// TwinCAT 3 PLC project PLC_1
// ProgramVersion: 3.1.4023.0
// libraries:
//   Tc2_ModbusRTU, * (Beckhoff Automation GmbH)
//   Tc2_Standard, * (Beckhoff Automation GmbH)
//   Tc2_System, * (Beckhoff Automation GmbH)
//   Tc3_Module, * (Beckhoff Automation GmbH)
// project tree:
//   / PlcTask.TcTTO
//   POUs/ MAIN.TcPOU, POU_Mdbus.TcPOU
// real-time tasks:
//   TASK PlcTask: cycle T#10ms, priority 20, ADS port 350

CONFIGURATION PLC_1
    RESOURCE PLC ON TwinCAT3
        TASK PlcTask(INTERVAL := T#10ms, PRIORITY := 20);
        PROGRAM MAIN WITH PlcTask : MAIN;
    END_RESOURCE
END_CONFIGURATION

// ---- POUs/MAIN.TcPOU
PROGRAM MAIN
VAR
END_VAR

POU_Mdbus();

END_PROGRAM

// ---- POUs/POU_Mdbus.TcPOU
PROGRAM POU_Mdbus
VAR
    fbModbusRead : FB_MBReadRegs ;
    fbModbusWrite : FB_MBWriteRegs ;
     
    iStep: INT;
     
    aModbusRead : ARRAY[1..10] OF INT ;
    aModbusWrite : ARRAY[1..10] OF INT ;    
END_VAR

CASE iStep OF
    0:
        fbModbusRead(bExecute:= FALSE );
        fbModbusWrite(bExecute := FALSE);       
        iStep := 10 ;
     
     
    10 : 
        fbModbusRead(
            sIPAddr:= '192.168.2.102', 
            nTCPPort:= 502, 
            nUnitID:= 255, 
            nQuantity:= 10, 
            nMBAddr:= 8000, 
            cbLength:= SIZEOF(aModbusRead), 
            pDestAddr:= ADR(aModbusRead), 
            bExecute:= TRUE, 
            tTimeout:= T#2S, 
            bBusy=> , 
            bError=> , 
            nErrId=> , 
            cbRead=> );
     
             
        IF  NOT fbModbusRead.bBusy THEN
            IF  NOT fbModbusRead.bError THEN 
                iStep := 20 ;
            ELSE
                iStep := 30 ;
            END_IF  
        END_IF
             
             
     
    20:
		iStep := 0;
     //  fbModbusWrite(
     //      sIPAddr:= '192.168.2.102', 
     //      nTCPPort:= 502, 
     //      nUnitID:= 1, 
     //      nQuantity:= 10, 
     //      nMBAddr:= 20, 
     //      cbLength:= SIZEOF(aModbusWrite), 
     //      pSrcAddr:= ADR(aModbusWrite), 
     //      bExecute:= TRUE, 
     //      tTimeout:= T#2S, 
     //      bBusy=> , 
     //      bError=> , 
     //      nErrId=> );
     //       
     //
     //  IF  NOT fbModbusWrite.bError OR fbModbusWrite.bBusy THEN
     //      iStep := 0 ;
     //  ELSE
     //      iStep := 30 ;
     //  END_IF
             
             
    30:
    ; //MODBUS READ ERROR
     
    31:
    ; //MODBUS WRITE ERROR
     
     
END_CASE

END_PROGRAM
